(* IEC 61131-3 sources: Elmo_Master/Lasal_PRG/Welcon8Axis_EtherCAT_Test_With_RobotAxis/Class/Robot_Handler, 1 file *)

(* ---- Robot_Handler.st ---- *)
(*!
<Class
	Name               = "Robot_Handler"
	Revision           = "0.0"
	RealtimeTask       = "false"
	CyclicTask         = "false"
	BackgroundTask     = "false"
	Sigmatek           = "false"
	OSInterface        = "false"
	HighPriority       = "false"
	Automatic          = "false"
	UpdateMode         = "Prescan"
	SharedCommandTable = "true"
	Objectsize         = "(420,120)">
	<Channels>
		<Server Name="Acc" Visualized="false" Initialize="true" DefValue="10 mm" WriteProtected="false" Retentive="File"/>
		<Server Name="ClassSvr" Visualized="false" Initialize="false" WriteProtected="true" Retentive="false"/>
		<Server Name="Jerk" Visualized="false" Initialize="true" DefValue="10 mm" WriteProtected="false" Retentive="File"/>
		<Server Name="Pos1" Visualized="false" Initialize="true" DefValue="100 mm" WriteProtected="false" Retentive="File"/>
		<Server Name="Pos2" Visualized="false" Initialize="true" DefValue="100 mm" WriteProtected="false" Retentive="File"/>
		<Server Name="Pos3" Visualized="false" Initialize="true" DefValue="100 mm" WriteProtected="false" Retentive="File"/>
		<Server Name="Pos4" Visualized="false" Initialize="true" DefValue="100 mm" WriteProtected="false" Retentive="File"/>
		<Server Name="Pos5" Visualized="false" Initialize="true" DefValue="100 mm" WriteProtected="false" Retentive="File"/>
		<Server Name="Pos6" Visualized="false" Initialize="true" DefValue="100 mm" WriteProtected="false" Retentive="File"/>
		<Server Name="Pos7" Visualized="false" Initialize="true" DefValue="100 mm" WriteProtected="false" Retentive="File"/>
		<Server Name="Pos8" Visualized="false" Initialize="true" DefValue="100 mm" WriteProtected="false" Retentive="File"/>
		<Server Name="PowerOff" Visualized="false" Initialize="false" WriteProtected="false" Retentive="false"/>
		<Server Name="PowerOn" Visualized="false" Initialize="false" WriteProtected="false" Retentive="false"/>
		<Server Name="RobotLock" Visualized="false" Initialize="false" WriteProtected="false" Retentive="false"/>
		<Server Name="RobotUnLock" Visualized="false" Initialize="false" WriteProtected="false" Retentive="false"/>
		<Server Name="Start" Visualized="false" Initialize="false" WriteProtected="false" Retentive="false"/>
		<Server Name="Stop" Visualized="false" Initialize="false" WriteProtected="false" Retentive="false"/>
		<Server Name="Velo" Visualized="false" Initialize="true" DefValue="10 mm" WriteProtected="false" Retentive="File"/>
		<Client Name="RobotBase" Required="true" Internal="false"/>
	</Channels>
</Class>
*)
Robot_Handler : CLASS
  //Servers:
	ClassSvr 	: SvrChCmd_DINT;
	PowerOn 	: SvrCh_DINT;
	PowerOff 	: SvrCh_DINT;
	RobotLock 	: SvrCh_DINT;
	RobotUnLock 	: SvrCh_DINT;
	Start 	: SvrCh_DINT;
	Stop 	: SvrCh_DINT;
	Pos1 	: SvrCh_DINT;
	Pos2 	: SvrCh_DINT;
	Pos3 	: SvrCh_DINT;
	Pos4 	: SvrCh_DINT;
	Pos5 	: SvrCh_DINT;
	Pos6 	: SvrCh_DINT;
	Pos7 	: SvrCh_DINT;
	Pos8 	: SvrCh_DINT;
	Velo 	: SvrCh_DINT;
	Acc 	: SvrCh_DINT;
	Jerk 	: SvrCh_DINT;
  //Clients:
	RobotBase 	: CltChCmd__LMCRobotBase;
  //Variables:
		Position 	: _LMCPROF_POS;
  //Functions:

	FUNCTION VIRTUAL GLOBAL PowerOn::Write
		VAR_INPUT
			input (EAX) 	: DINT;
		END_VAR
		VAR_OUTPUT
			result (EAX) 	: DINT;
		END_VAR;

	FUNCTION VIRTUAL GLOBAL PowerOff::Write
		VAR_INPUT
			input (EAX) 	: DINT;
		END_VAR
		VAR_OUTPUT
			result (EAX) 	: DINT;
		END_VAR;

	FUNCTION VIRTUAL GLOBAL RobotLock::Write
		VAR_INPUT
			input (EAX) 	: DINT;
		END_VAR
		VAR_OUTPUT
			result (EAX) 	: DINT;
		END_VAR;

	FUNCTION VIRTUAL GLOBAL RobotUnLock::Write
		VAR_INPUT
			input (EAX) 	: DINT;
		END_VAR
		VAR_OUTPUT
			result (EAX) 	: DINT;
		END_VAR;

	FUNCTION VIRTUAL GLOBAL Start::Write
		VAR_INPUT
			input (EAX) 	: DINT;
		END_VAR
		VAR_OUTPUT
			result (EAX) 	: DINT;
		END_VAR;

	FUNCTION VIRTUAL GLOBAL Stop::Write
		VAR_INPUT
			input (EAX) 	: DINT;
		END_VAR
		VAR_OUTPUT
			result (EAX) 	: DINT;
		END_VAR;
  //Tables:
	FUNCTION @STD
		VAR_OUTPUT
			ret_code	: CONFSTATES;
		END_VAR;
	FUNCTION GLOBAL TAB @CT_;
END_CLASS;

#pragma usingLtd _LMCRobotBase

FUNCTION VIRTUAL GLOBAL Robot_Handler::PowerOn::Write
	VAR_INPUT
		input (EAX) 	: DINT;
	END_VAR
	VAR_OUTPUT
		result (EAX) 	: DINT;
	END_VAR

	PowerOn := input;
  RobotBase.RobotOn(Mode:=_LMCRobotBase::_ACTIVE);
	result := PowerOn;

END_FUNCTION

FUNCTION VIRTUAL GLOBAL Robot_Handler::PowerOff::Write
	VAR_INPUT
		input (EAX) 	: DINT;
	END_VAR
	VAR_OUTPUT
		result (EAX) 	: DINT;
	END_VAR

	PowerOff := input;
  RobotBase.RobotOff();
	result := PowerOff;

END_FUNCTION

FUNCTION VIRTUAL GLOBAL Robot_Handler::RobotLock::Write
	VAR_INPUT
		input (EAX) 	: DINT;
	END_VAR
	VAR_OUTPUT
		result (EAX) 	: DINT;
	END_VAR

	RobotLock := input;
  RobotBase.LockProfile(Axis1:=1, Axis2:=1, Axis3:=1, Axis4:=1, Axis5:=1, Axis6:=1, Axis7:=1, Axis8:=1, Axis9:=0);
	result := RobotLock;

END_FUNCTION

FUNCTION VIRTUAL GLOBAL Robot_Handler::RobotUnLock::Write
	VAR_INPUT
		input (EAX) 	: DINT;
	END_VAR
	VAR_OUTPUT
		result (EAX) 	: DINT;
	END_VAR

	RobotUnLock := input;
  RobotBase.UnlockProfile();
	result := RobotUnLock;

END_FUNCTION

FUNCTION VIRTUAL GLOBAL Robot_Handler::Start::Write
	VAR_INPUT
		input (EAX) 	: DINT;
	END_VAR
	VAR_OUTPUT
		result (EAX) 	: DINT;
	END_VAR

	Start := input;

  Position.Pos1 := Pos1;
  Position.Pos2 := Pos2;
  Position.Pos3 := Pos3;
  Position.Pos4 := Pos4;
  Position.Pos5 := Pos5;
  Position.Pos6 := Pos6;
  Position.Pos7 := Pos7;
  Position.Pos8 := Pos8;

  RobotBase.MoveLinear(pPositions:=#Position,
                       CmdConfig:=0,
                       Velocity:=Velo,
                       Accel:=Acc,
                       Decel:=Acc,
                       TransMode:=_LMCPROF_EXACT_STOP,
                       TransRadius:=0,
                       Jerk:=Jerk);
	result := Start;

END_FUNCTION

FUNCTION VIRTUAL GLOBAL Robot_Handler::Stop::Write
	VAR_INPUT
		input (EAX) 	: DINT;
	END_VAR
	VAR_OUTPUT
		result (EAX) 	: DINT;
	END_VAR

	Stop := input;
  RobotBase.StopMove(Mode:=3, Decel:=Acc, Jerk:=Jerk);
	result := Stop;

END_FUNCTION
